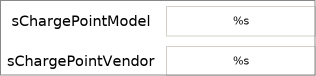
VISUALIZATION Visu_BootNotification  // 316x76
VAR_IN_OUT
	fbStation 		: FB_Station;
END_VAR
    Textfield (166,6 150x30), "%s", text variable: fbStation._stVisu.stBoot.sChargePointModel
    Textfield (166,46 150x30), "%s", text variable: fbStation._stVisu.stBoot.sChargePointVendor
    Label (6,6 150x30), "sChargePointModel"
    Label (6,46 150x30), "sChargePointVendor"
END_VISUALIZATION

(* stored: Version 1.1.0.1
   Visu Visu_BootNotification: Id {49058733-0733-4db9-b7ce-79c92f7c0085} *)
